// TIA Portal V19 export
TYPE "LEXCHANGETRAY_typeVfdInterface"
// commandConfiguration: LBC_typeSinaSpeedCommandConfiguration
// commands: LBC_typeSinaSpeedManualCommands
// monitoring: LEXCHANGETRAY_typeVfdProcessValues
// configuration: LBC_typeSinaSpeedConfiguration
// stored: Access Published
   STRUCT
      commandConfiguration : "LBC_typeSinaSpeedCommandConfiguration";
      commands : "LBC_typeSinaSpeedManualCommands";
      monitoring { S7_SetPoint := 'True'} : "LEXCHANGETRAY_typeVfdProcessValues";
      configuration : "LBC_typeSinaSpeedConfiguration";
   END_STRUCT;
END_TYPE
